FUNCTION_BLOCK FB_SimpleLinearTwoWayDrive
VAR_INPUT
	SensorHomePos: BOOL;
	SensorWorkPos: BOOL;
	Enable: BOOL;
	LockHomePos: BOOL;
	LockWorkPos: BOOL;
	HoldPosition: BOOL;	// TRUE: Hold output to true even if position has been reached
	ToHome: BOOL;
	ToWork: BOOL;
END_VAR
VAR_OUTPUT	
	ActorHomePos: BOOL;
	ActorWorkPos: BOOL;
END_VAR
VAR
END_VAR

ActorHomePos := SetOutput(ToHome, SensorHomePos, LockHomePos, ActorWorkPos);
ActorWorkPos := SetOutput(ToWork, SensorWorkPos, LockWorkPos, ActorHomePos);

METHOD PRIVATE SetOutput : BOOL
VAR_INPUT
	MoveToPos : BOOL;
	PosReached: BOOL;
	DirectionLocked: BOOL;
	OutputInterlock: BOOL;
END_VAR
SetOutput := MoveToPos AND Enable AND NOT DirectionLocked AND NOT OutputInterlock AND (NOT PosReached OR HoldPosition);
END_METHOD

END_FUNCTION_BLOCK

(* stored: Version 1.1.0.1, ProductVersion 3.1.4024.11
   POU FB_SimpleLinearTwoWayDrive: Id {d5079cf3-2029-4674-b5d0-714b53c5075a}, SpecialFunc None
   Method SetOutput: Id {2b2cbc49-cd42-42ab-8144-70652882f6fc} *)
